// TIA Portal project "DADKLT" (V16)

(* hardware
DEVICE "S7-1200 station_1"  S7-1200 Station
   slot 0: "Rack_0"  S7-1200 Rack  Rack  V1.0
   slot 1: "PLC_1"  CPU 1214C DC/DC/DC  6ES7 214-1AG40-0XB0  V4.4
DEVICE "PC-System_1"  SIMATIC PC station
   slot 0: "SIMATIC PC station"  Rail  SIMATIC PC-Station  V1.0
      slot 125: "Stationmanager"  Station_Manager  V6.0.4
   slot 1: "HMI_RT_1"  WinCC RT Advanced  6AV2 104-0xxxx-xxxx  16.0.0.0
      slot 33792: "Computer interface"  Host interface
   slot 2: "IE general_1"  IE General  IE_CP  V8.2.0
*)

// ===== PLC "PLC_1"  CPU 1214C DC/DC/DC =====

VAR_GLOBAL   // PLC tag table "Default tag table"
   "LEVEL_TANK" AT %IW32 : Int;
   "ACTUAL_LEVEL_TANK" AT %MD0 : Real;
   "PID_SET_POINT" AT %MD4 : Real;
   "FILLING VALUE" AT %MW8 : Int;
   "OPEN_ACTUATOR" AT %QW30 : Int;
   "ENABLE_PID" AT %M10.0 : Bool;
END_VAR

FUNCTION "MHJ-PLC-Lab-Function-S71200" : Void   // FC9000, SCL
{ S7_Optimized_Access := 'TRUE' }
VERSION : 0.1
   VAR_TEMP
      rdTimeReturn : Int;
      outputTime : DTL;
      SyncVal : Byte;
      forVal : Int;
      forVal_2 : Int;
      Value : Byte;
   END_VAR
   VAR CONSTANT
      CompVal : Byte := 16#34;
      Value_01 : Byte := 16#11;
      Value_01_DW : DWord := 16#A165_D992;
      Value_02_DW : DWord := 16#58BE_4401;
   END_VAR
BEGIN

   #Value:=PEEK(area := 16#82,
        dbNumber := 0,
        byteOffset := 511);
   #Value := #Value + 1;

   POKE(area := 16#82,
        dbNumber := 0,
        byteOffset := 511,
        value := #Value);

   POKE(area:=16#81,
        dbNumber:=0,
        byteOffset:=1016,
        value:=#Value_01_DW);
   POKE(area := 16#81,
        dbNumber := 0,
        byteOffset := 1020,
        value := #Value_02_DW);

   POKE(area := 16#81,
        dbNumber := 0,
        byteOffset := 511,
        value := B#16#00);

   FOR #forVal := 0 TO 120 DO
       FOR #forVal_2:=0 TO 10 DO
           #rdTimeReturn:=RD_SYS_T(#outputTime);
           #rdTimeReturn := WR_SYS_T(#outputTime);
           #rdTimeReturn := RD_SYS_T(#outputTime);
           #rdTimeReturn := WR_SYS_T(#outputTime);
       END_FOR;
       #SyncVal:= PEEK(area := 16#81,
                      dbNumber := 0,
                      byteOffset := 511);
       IF #SyncVal = #CompVal THEN
          GOTO M_1;
       END_IF;
   END_FOR;
   RETURN;

   M_1:
   POKE(area := 16#81,
        dbNumber := 0,
        byteOffset := 511,
        value := B#16#0);
END_FUNCTION

ORGANIZATION_BLOCK "Main"   // OB1, LAD, ProgramCycle
TITLE = "Main Program Sweep (Cycle)"
{ S7_Optimized_Access := 'TRUE' }
VERSION : 0.1
   VAR_INPUT
      Initial_Call : Bool;   // Initial call of this OB
      Remanence : Bool;   // =True, if remanent data are available
   END_VAR
   VAR_TEMP
      Temp1 : Real;
   END_VAR
BEGIN

REGION Network 1
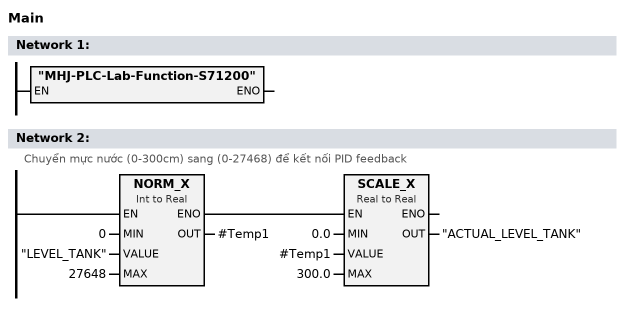
   RUNG wire#powerrail
      "MHJ-PLC-Lab-Function-S71200"()
   END_RUNG
   // the same network as SCL:
   "MHJ-PLC-Lab-Function-S71200"();
END_REGION

REGION Network 2
   // Chuyển mực nước (0-300cm) sang (0-27468) để kết nối PID feedback
   RUNG wire#powerrail
      { S7_Templates := "[SrcType := Int, DestType := Real]" } Normalize(min := 0, value := "LEVEL_TANK", max := 27648, out => #Temp1)
      { S7_Templates := "[SrcType := Real, DestType := Real]" } Scale(min := 0.0, value := #Temp1, max := 300.0, out => "ACTUAL_LEVEL_TANK")
   END_RUNG
   // the same network as SCL:
   #Temp1 := NORM_X(MIN := 0, VALUE := "LEVEL_TANK", MAX := 27648);
   "ACTUAL_LEVEL_TANK" := SCALE_X(MIN := 0.0, VALUE := #Temp1, MAX := 300.0);
END_REGION
END_ORGANIZATION_BLOCK

ORGANIZATION_BLOCK "Cyclic interrupt"   // OB30, LAD, CyclicInterrupt
{ S7_Optimized_Access := 'TRUE' }
VERSION : 0.1
   VAR_INPUT
      Initial_Call : Bool;   // Initial call of this OB
      Event_Count : Int;   // Events discarded
   END_VAR
   VAR_TEMP   // added for the SCL form of the ladder/FBD networks
      _w1 : Bool;
   END_VAR
BEGIN

REGION Network 1
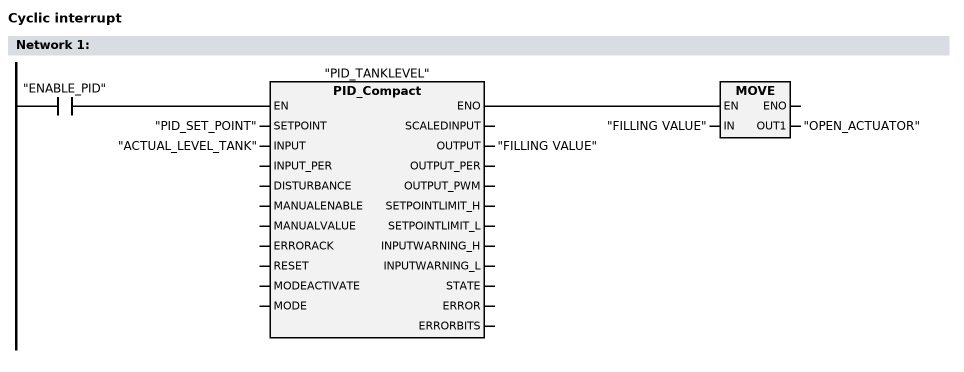
   // ENO of a box is taken as its EN; it also drops when the box reports an error
   #_w1 := "ENABLE_PID";
   IF #_w1 THEN
       "PID_TANKLEVEL"(Setpoint := "PID_SET_POINT", Input := "ACTUAL_LEVEL_TANK", Output => "FILLING VALUE");   // PID_Compact
       "OPEN_ACTUATOR" := "FILLING VALUE";
   END_IF;
END_REGION
END_ORGANIZATION_BLOCK

(* ===== HMI "HMI_RT_1" =====
system functions are stored by id; their names below are inferred from use
connection "HMI_Connection_1": ETHERNET, S7_1200_OMS

HMI tags "Default tag table"
   "PID_SET_POINT" : Real = PLC PID_SET_POINT AT %MD4, 1 s
   "ACTUAL_LEVEL_TANK" : Real = PLC ACTUAL_LEVEL_TANK AT %MD0, 1 s
   "ENABLE_PID" : Bool = PLC ENABLE_PID AT %M10.0, 1 s
   "OPEN_ACTUATOR" : Int = PLC OPEN_ACTUATOR AT %QW30, 1 s
   "PID_TANKLEVEL_CtrlParamsBackUp_Gain" : Real = PLC PID_TANKLEVEL.CtrlParamsBackUp.Gain, 1 s
   "PID_TANKLEVEL_CtrlParamsBackUp_Ti" : Real = PLC PID_TANKLEVEL.CtrlParamsBackUp.Ti, 1 s
   "PID_TANKLEVEL_CtrlParamsBackUp_Td" : Real = PLC PID_TANKLEVEL.CtrlParamsBackUp.Td, 1 s
   "PID_TANKLEVEL_Output" : Real = PLC PID_TANKLEVEL.Output, 1 s

screen "PID SCREEN" 1024x768
   TextField "Text field_1" at 0,1 size 298x59; Text 'ĐỒ ÁN ĐIỀU KHIỂN LẬP TRÌNH'
   TextField "Text field_4" at 295,1 size 505x59; Text 'MỔ PHỎNG ĐIỀU KHIỂN PID VỚI FACOTRY IO'
   TextField "Text field_2" at 798,0 size 226x59; Text 'ĐÀO BẢO TÍN - 20151230'
   IOField "I/O field_1" at 77,176 size 133x43; FormatPattern 999.9
      ProcessValue <- "PID_SET_POINT"
   TextField "Text field_3" at 4,178 size 48x42; Text 'SP'
   TextField "Text field_5" at 204,176 size 59x42; Text 'CM'
   IOField "I/O field_2" at 77,237 size 133x43; FormatPattern 999.9
      ProcessValue <- "ACTUAL_LEVEL_TANK"
   TextField "Text field_6" at 4,237 size 54x42; Text 'PV'
   Button "Button_1" at 7,75 size 232x83; TextOff 'ENABLE PID SYSTEM'
      on Click: InvertBit("ENABLE_PID")
      Appearance <- "ENABLE_PID"
   TrendView "Trend view_1" at 271,82 size 747x496
   IOField "I/O field_3" at 77,413 size 132x43; FormatPattern 999.9
      ProcessValue <- "PID_TANKLEVEL_CtrlParamsBackUp_Gain"
   TextField "Text field_8" at 4,413 size 61x42; Text 'GAIN'
   IOField "I/O field_4" at 77,474 size 130x43; FormatPattern 999.9
      ProcessValue <- "PID_TANKLEVEL_CtrlParamsBackUp_Ti"
   IOField "I/O field_5" at 77,534 size 130x43; FormatPattern 999.9
      ProcessValue <- "PID_TANKLEVEL_CtrlParamsBackUp_Td"
   TextField "Text field_9" at 4,467 size 56x42; Text 'Ti'
   TextField "Text field_10" at 4,537 size 58x42; Text 'Td'
   TextField "Text field_11" at 12,357 size 224x41; Text 'PID Adjustment'
   TextField "Text field_7" at 204,240 size 59x42; Text 'CM'
   TextField "Text field_12" at 4,310 size 54x42; Text 'OUT'
   IOField "I/O field_6" at 77,309 size 133x43; FormatPattern 999.9
      ProcessValue <- "PID_TANKLEVEL_Output"
   TextField "Text field_13" at 204,307 size 59x42; Text '%'
*)